// Mitsubishi GX Works2 project: Step Control(end)   PLC: Q01U

PROGRAM conveyor
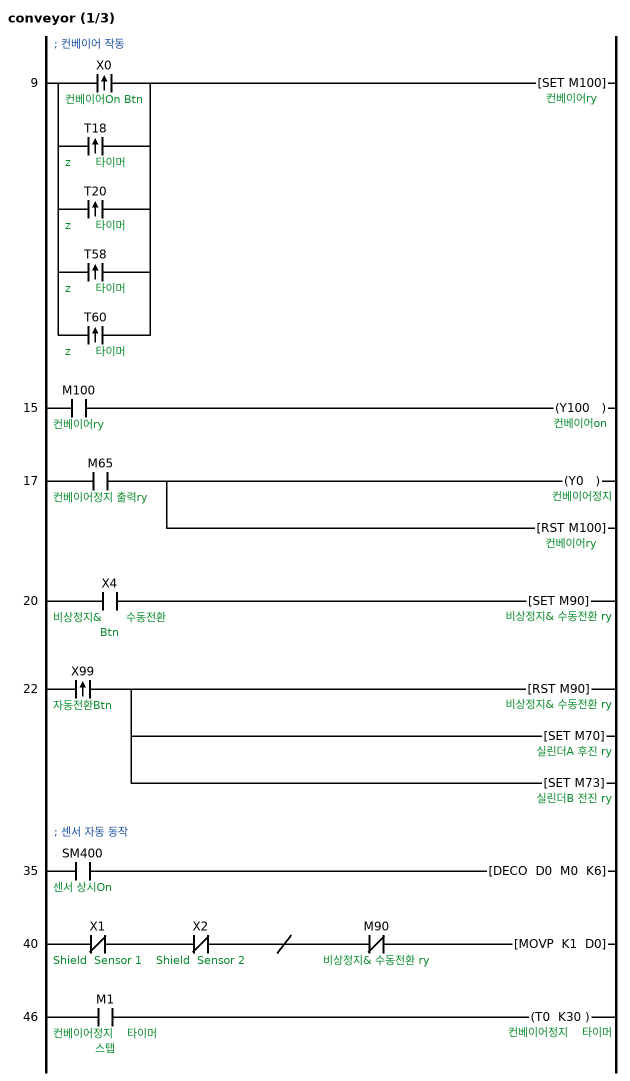
; 컨베이어 작동
9     LDP     X0  ; 컨베이어On Btn
      ORP     T18  ; z       타이머
      ORP     T20  ; z       타이머
      ORP     T58  ; z       타이머
      ORP     T60  ; z       타이머
      SET     M100  ; 컨베이어ry
15    LD      M100  ; 컨베이어ry
      OUT     Y100  ; 컨베이어on
17    LD      M65  ; 컨베이어정지 출력ry
      OUT     Y0  ; 컨베이어정지
      RST     M100  ; 컨베이어ry
20    LD      X4  ; 비상정지&       수동전환 Btn
      SET     M90  ; 비상정지& 수동전환 ry
22    LDP     X99  ; 자동전환Btn
      RST     M90  ; 비상정지& 수동전환 ry
      SET     M70  ; 실린더A 후진 ry
      SET     M73  ; 실린더B 전진 ry
; 센서 자동 동작
35    LD      SM400  ; 센서 상시On
      DECO    D0 M0 K6
40    LDI     X1  ; Shield  Sensor 1
      ANI     X2  ; Shield  Sensor 2
      INV
      ANI     M90  ; 비상정지& 수동전환 ry
      MOVP    K1 D0
46    LD      M1  ; 컨베이어정지    타이머  스탭
      OUT     T0 K30  ; 컨베이어정지    타이머
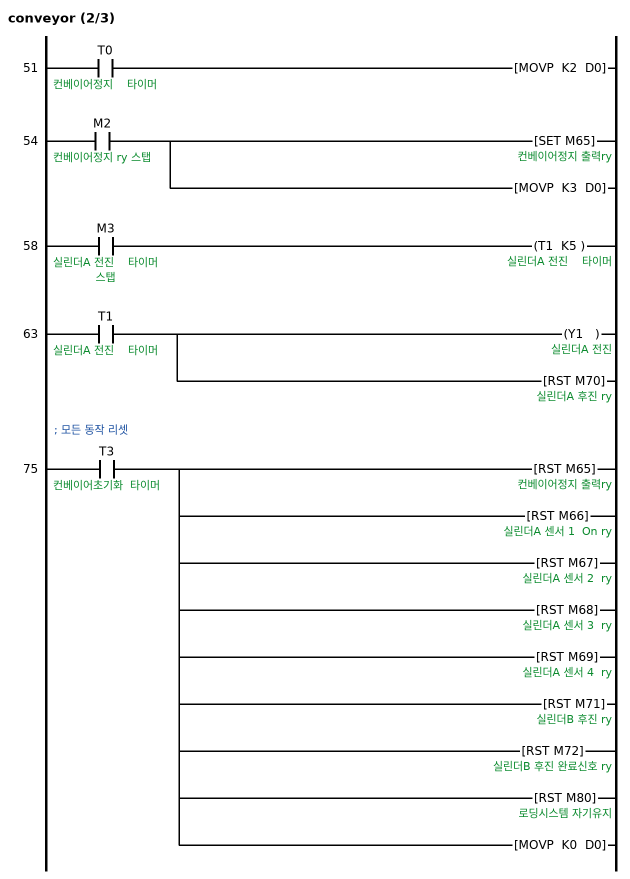
51    LD      T0  ; 컨베이어정지    타이머
      MOVP    K2 D0
54    LD      M2  ; 컨베이어정지 ry 스탭
      SET     M65  ; 컨베이어정지 출력ry
      MOVP    K3 D0
58    LD      M3  ; 실린더A 전진    타이머  스탭
      OUT     T1 K5  ; 실린더A 전진    타이머
63    LD      T1  ; 실린더A 전진    타이머
      OUT     Y1  ; 실린더A 전진
      RST     M70  ; 실린더A 후진 ry
; 모든 동작 리셋
75    LD      T3  ; 컨베이어초기화  타이머
      RST     M65  ; 컨베이어정지 출력ry
      RST     M66  ; 실린더A 센서 1  On ry
      RST     M67  ; 실린더A 센서 2  ry
      RST     M68  ; 실린더A 센서 3  ry
      RST     M69  ; 실린더A 센서 4  ry
      RST     M71  ; 실린더B 후진 ry
      RST     M72  ; 실린더B 후진 완료신호 ry
      RST     M80  ; 로딩시스템 자기유지
      MOVP    K0 D0
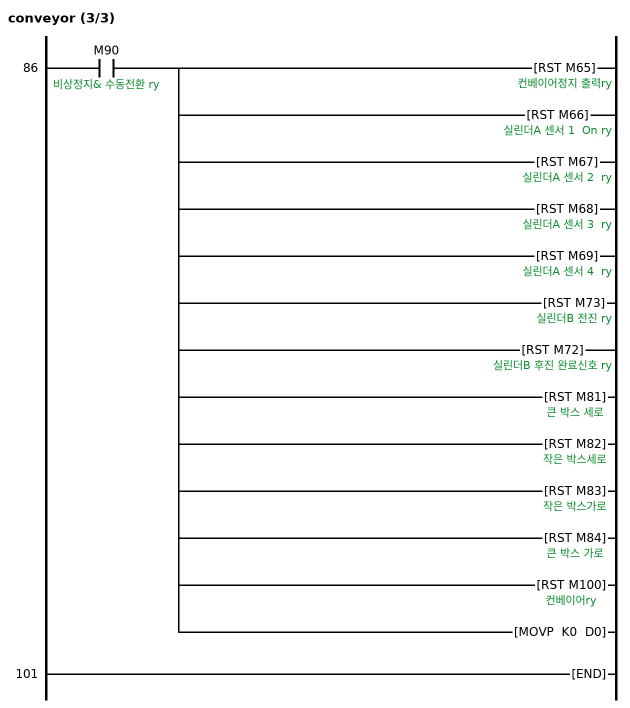
86    LD      M90  ; 비상정지& 수동전환 ry
      RST     M65  ; 컨베이어정지 출력ry
      RST     M66  ; 실린더A 센서 1  On ry
      RST     M67  ; 실린더A 센서 2  ry
      RST     M68  ; 실린더A 센서 3  ry
      RST     M69  ; 실린더A 센서 4  ry
      RST     M73  ; 실린더B 전진 ry
      RST     M72  ; 실린더B 후진 완료신호 ry
      RST     M81  ; 큰 박스 세로
      RST     M82  ; 작은 박스세로
      RST     M83  ; 작은 박스가로
      RST     M84  ; 큰 박스 가로
      RST     M100  ; 컨베이어ry
      MOVP    K0 D0
101   END
END_PROGRAM

PROGRAM cylinder
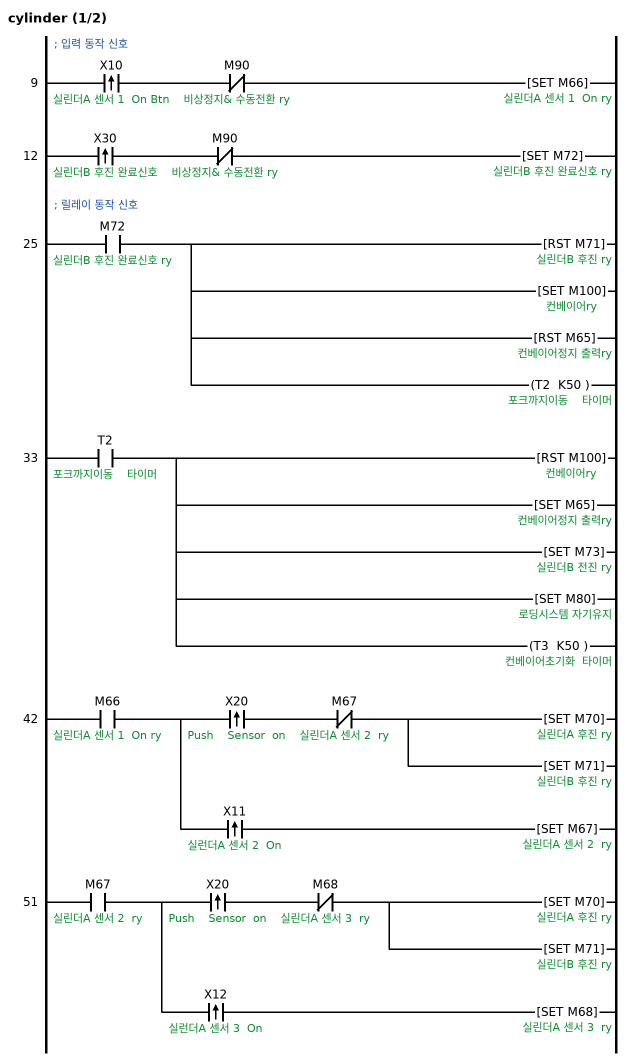
; 입력 동작 신호
9     LDP     X10  ; 실린더A 센서 1  On Btn
      ANI     M90  ; 비상정지& 수동전환 ry
      SET     M66  ; 실린더A 센서 1  On ry
12    LDP     X30  ; 실린더B 후진 완료신호
      ANI     M90  ; 비상정지& 수동전환 ry
      SET     M72  ; 실린더B 후진 완료신호 ry
; 릴레이 동작 신호
25    LD      M72  ; 실린더B 후진 완료신호 ry
      RST     M71  ; 실린더B 후진 ry
      SET     M100  ; 컨베이어ry
      RST     M65  ; 컨베이어정지 출력ry
      OUT     T2 K50  ; 포크까지이동    타이머
33    LD      T2  ; 포크까지이동    타이머
      RST     M100  ; 컨베이어ry
      SET     M65  ; 컨베이어정지 출력ry
      SET     M73  ; 실린더B 전진 ry
      SET     M80  ; 로딩시스템 자기유지
      OUT     T3 K50  ; 컨베이어초기화  타이머
42    LD      M66  ; 실린더A 센서 1  On ry
      MPS
      ANDP    X20  ; Push    Sensor  on
      ANI     M67  ; 실린더A 센서 2  ry
      SET     M70  ; 실린더A 후진 ry
      SET     M71  ; 실린더B 후진 ry
      MPP
      ANDP    X11  ; 실런더A 센서 2  On
      SET     M67  ; 실린더A 센서 2  ry
51    LD      M67  ; 실린더A 센서 2  ry
      MPS
      ANDP    X20  ; Push    Sensor  on
      ANI     M68  ; 실린더A 센서 3  ry
      SET     M70  ; 실린더A 후진 ry
      SET     M71  ; 실린더B 후진 ry
      MPP
      ANDP    X12  ; 실런더A 센서 3  On
      SET     M68  ; 실린더A 센서 3  ry
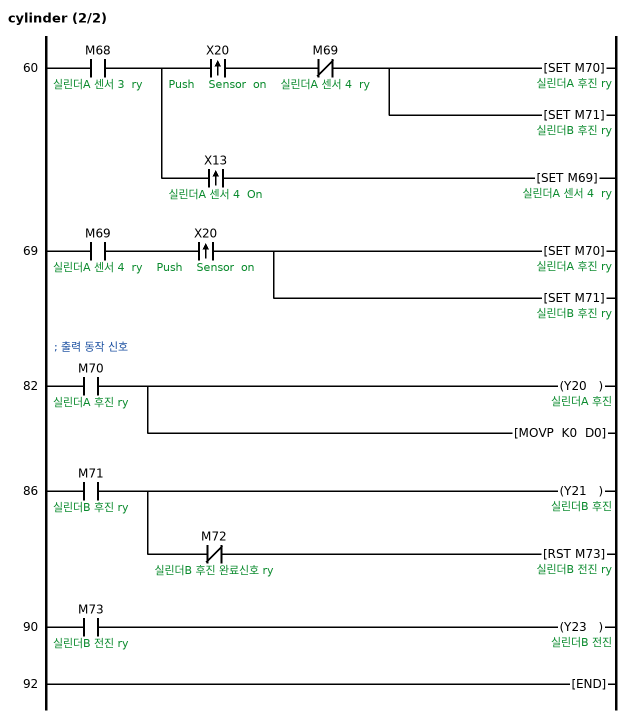
60    LD      M68  ; 실린더A 센서 3  ry
      MPS
      ANDP    X20  ; Push    Sensor  on
      ANI     M69  ; 실린더A 센서 4  ry
      SET     M70  ; 실린더A 후진 ry
      SET     M71  ; 실린더B 후진 ry
      MPP
      ANDP    X13  ; 실린더A 센서 4  On
      SET     M69  ; 실린더A 센서 4  ry
69    LD      M69  ; 실린더A 센서 4  ry
      ANDP    X20  ; Push    Sensor  on
      SET     M70  ; 실린더A 후진 ry
      SET     M71  ; 실린더B 후진 ry
; 출력 동작 신호
82    LD      M70  ; 실린더A 후진 ry
      OUT     Y20  ; 실린더A 후진
      MOVP    K0 D0
86    LD      M71  ; 실린더B 후진 ry
      OUT     Y21  ; 실린더B 후진
      ANI     M72  ; 실린더B 후진 완료신호 ry
      RST     M73  ; 실린더B 전진 ry
90    LD      M73  ; 실린더B 전진 ry
      OUT     Y23  ; 실린더B 전진
92    END
END_PROGRAM

PROGRAM manual
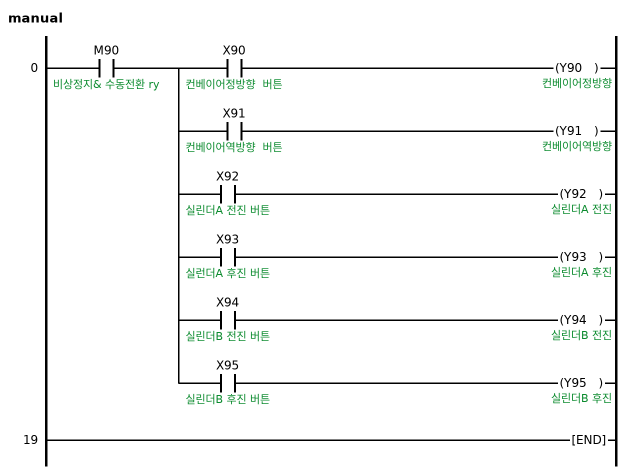
0     LD      M90  ; 비상정지& 수동전환 ry
      MPS
      AND     X90  ; 컨베이어정방향  버튼
      OUT     Y90  ; 컨베이어정방향
      MRD
      AND     X91  ; 컨베이어역방향  버튼
      OUT     Y91  ; 컨베이어역방향
      MRD
      AND     X92  ; 실린더A 전진 버튼
      OUT     Y92  ; 실린더A 전진
      MRD
      AND     X93  ; 실런더A 후진 버튼
      OUT     Y93  ; 실린더A 후진
      MRD
      AND     X94  ; 실린더B 전진 버튼
      OUT     Y94  ; 실린더B 전진
      MPP
      AND     X95  ; 실린더B 후진 버튼
      OUT     Y95  ; 실린더B 후진
19    END
END_PROGRAM

PROGRAM boxSize
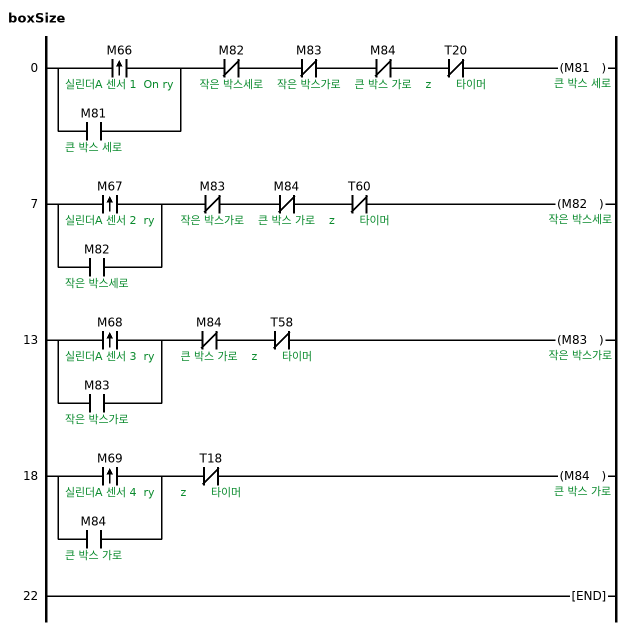
0     LDP     M66  ; 실린더A 센서 1  On ry
      OR      M81  ; 큰 박스 세로
      ANI     M82  ; 작은 박스세로
      ANI     M83  ; 작은 박스가로
      ANI     M84  ; 큰 박스 가로
      ANI     T20  ; z       타이머
      OUT     M81  ; 큰 박스 세로
7     LDP     M67  ; 실린더A 센서 2  ry
      OR      M82  ; 작은 박스세로
      ANI     M83  ; 작은 박스가로
      ANI     M84  ; 큰 박스 가로
      ANI     T60  ; z       타이머
      OUT     M82  ; 작은 박스세로
13    LDP     M68  ; 실린더A 센서 3  ry
      OR      M83  ; 작은 박스가로
      ANI     M84  ; 큰 박스 가로
      ANI     T58  ; z       타이머
      OUT     M83  ; 작은 박스가로
18    LDP     M69  ; 실린더A 센서 4  ry
      OR      M84  ; 큰 박스 가로
      ANI     T18  ; z       타이머
      OUT     M84  ; 큰 박스 가로
22    END
END_PROGRAM

PROGRAM Box4move
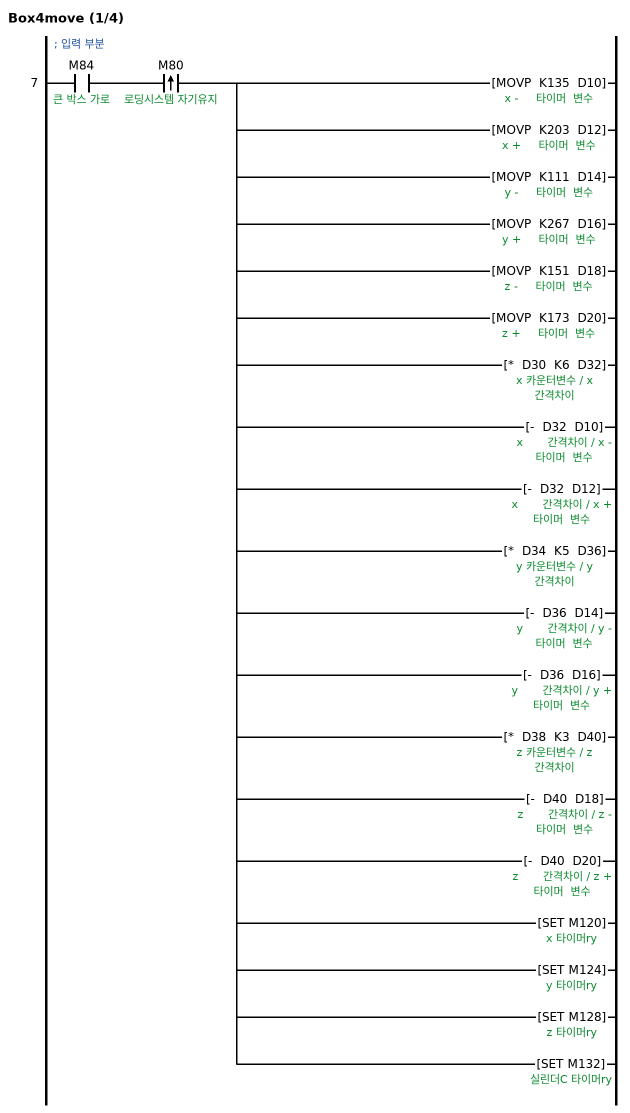
; 입력 부분
7     LD      M84  ; 큰 박스 가로
      ANDP    M80  ; 로딩시스템 자기유지
      MOVP    K135 D10  ; x -     타이머  변수
      MOVP    K203 D12  ; x +     타이머  변수
      MOVP    K111 D14  ; y -     타이머  변수
      MOVP    K267 D16  ; y +     타이머  변수
      MOVP    K151 D18  ; z -     타이머  변수
      MOVP    K173 D20  ; z +     타이머  변수
      *       D30 K6 D32  ; x 카운터변수 / x       간격차이
      -       D32 D10
      -       D32 D12
      *       D34 K5 D36  ; y 카운터변수 / y       간격차이
      -       D36 D14
      -       D36 D16
      *       D38 K3 D40  ; z 카운터변수 / z       간격차이
      -       D40 D18
      -       D40 D20
      SET     M120  ; x 타이머ry
      SET     M124  ; y 타이머ry
      SET     M128  ; z 타이머ry
      SET     M132  ; 실린더C 타이머ry
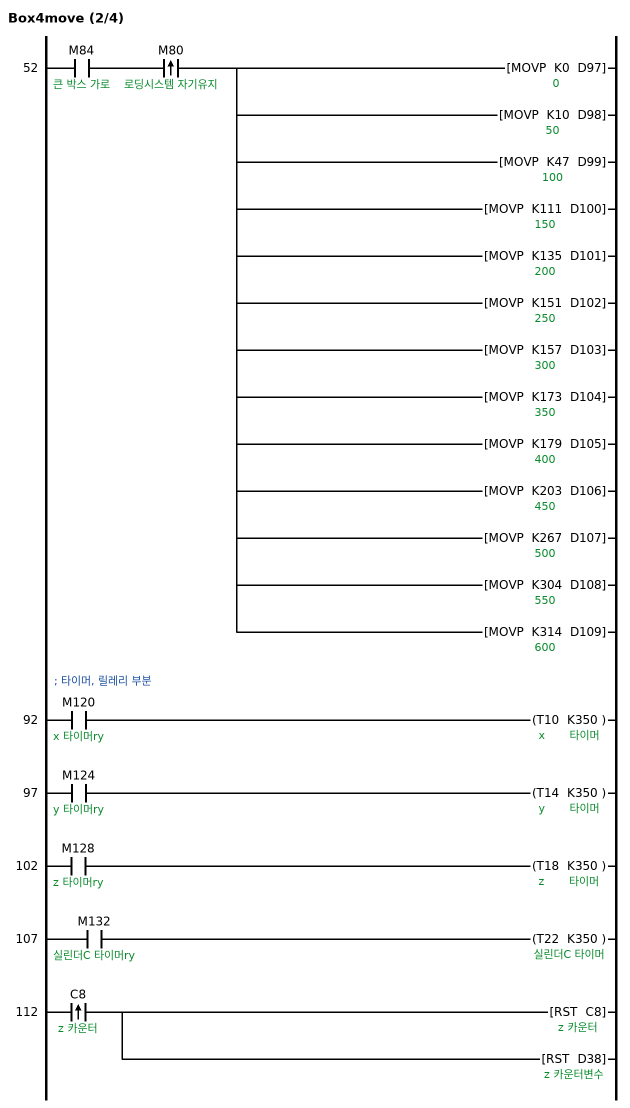
52    LD      M84  ; 큰 박스 가로
      ANDP    M80  ; 로딩시스템 자기유지
      MOVP    K0 D97  ; 0
      MOVP    K10 D98  ; 50
      MOVP    K47 D99  ; 100
      MOVP    K111 D100  ; 150
      MOVP    K135 D101  ; 200
      MOVP    K151 D102  ; 250
      MOVP    K157 D103  ; 300
      MOVP    K173 D104  ; 350
      MOVP    K179 D105  ; 400
      MOVP    K203 D106  ; 450
      MOVP    K267 D107  ; 500
      MOVP    K304 D108  ; 550
      MOVP    K314 D109  ; 600
; 타이머, 릴레리 부분
92    LD      M120  ; x 타이머ry
      OUT     T10 K350  ; x       타이머
97    LD      M124  ; y 타이머ry
      OUT     T14 K350  ; y       타이머
102   LD      M128  ; z 타이머ry
      OUT     T18 K350  ; z       타이머
107   LD      M132  ; 실린더C 타이머ry
      OUT     T22 K350  ; 실린더C 타이머
112   LDP     C8  ; z 카운터
      RST     C8  ; z 카운터
      RST     D38  ; z 카운터변수
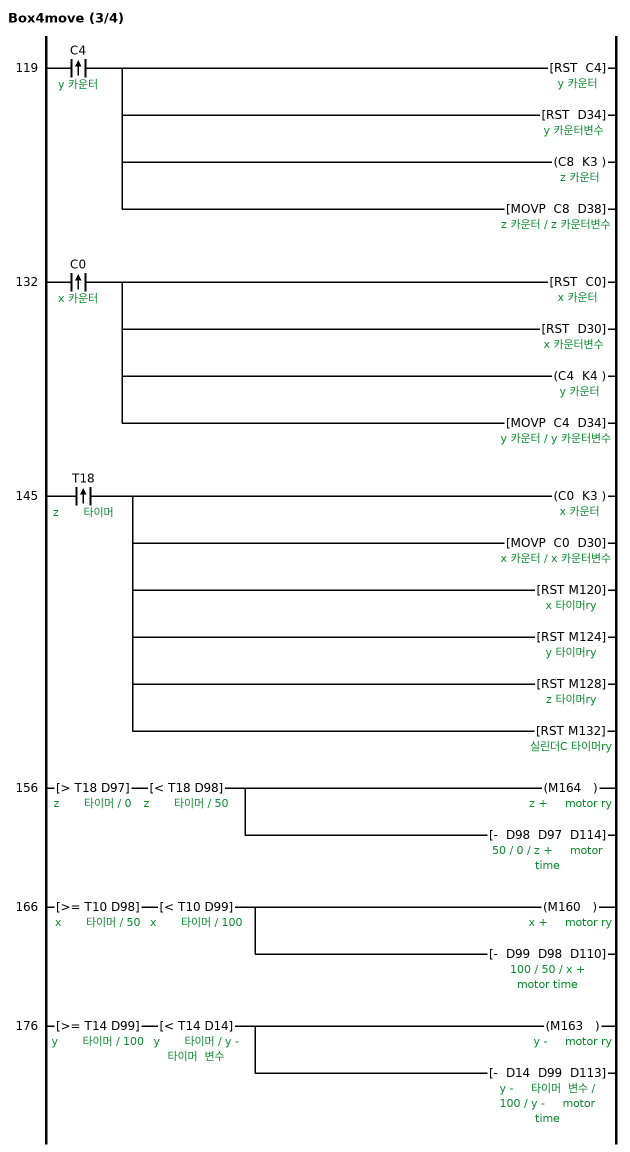
119   LDP     C4  ; y 카운터
      RST     C4  ; y 카운터
      RST     D34  ; y 카운터변수
      OUT     C8 K3  ; z 카운터
      MOVP    C8 D38
132   LDP     C0  ; x 카운터
      RST     C0  ; x 카운터
      RST     D30  ; x 카운터변수
      OUT     C4 K4  ; y 카운터
      MOVP    C4 D34
145   LDP     T18  ; z       타이머
      OUT     C0 K3  ; x 카운터
      MOVP    C0 D30
      RST     M120  ; x 타이머ry
      RST     M124  ; y 타이머ry
      RST     M128  ; z 타이머ry
      RST     M132  ; 실린더C 타이머ry
156   LD>     T18 D97  ; z       타이머 / 0
      AND<    T18 D98  ; z       타이머 / 50
      OUT     M164  ; z +     motor ry
      -       D98 D97 D114  ; z +     motor time
166   LD>=    T10 D98  ; x       타이머 / 50
      AND<    T10 D99  ; x       타이머 / 100
      OUT     M160  ; x +     motor ry
      -       D99 D98 D110  ; x +     motor time
176   LD>=    T14 D99  ; y       타이머 / 100
      AND<    T14 D14  ; y       타이머 / y -     타이머  변수
      OUT     M163  ; y -     motor ry
      -       D14 D99 D113  ; y -     motor time
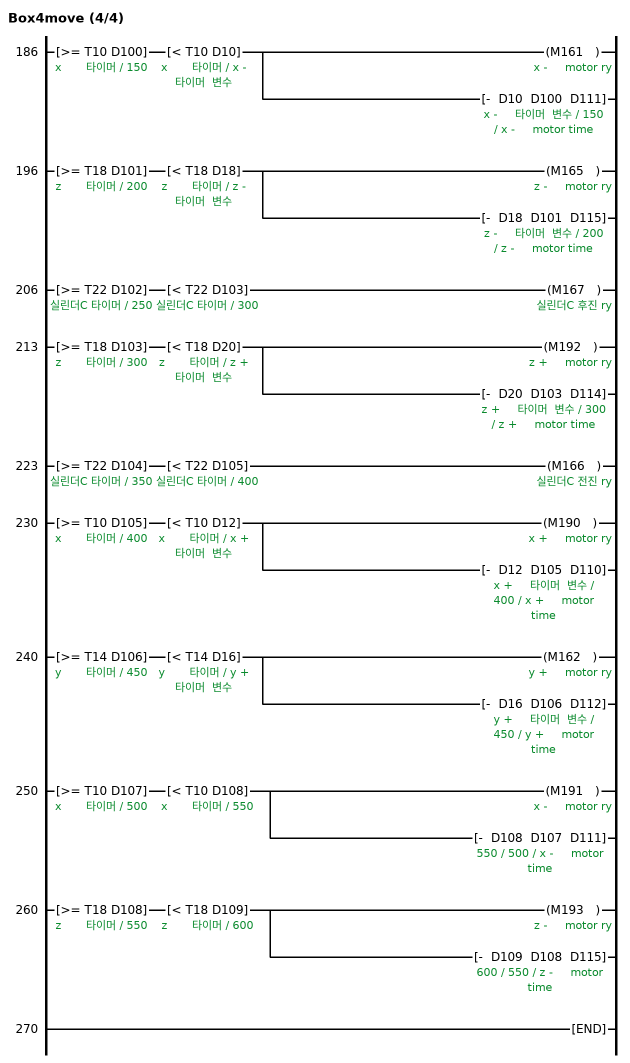
186   LD>=    T10 D100  ; x       타이머 / 150
      AND<    T10 D10  ; x       타이머 / x -     타이머  변수
      OUT     M161  ; x -     motor ry
      -       D10 D100 D111  ; x -     motor time
196   LD>=    T18 D101  ; z       타이머 / 200
      AND<    T18 D18  ; z       타이머 / z -     타이머  변수
      OUT     M165  ; z -     motor ry
      -       D18 D101 D115  ; z -     motor time
206   LD>=    T22 D102  ; 실린더C 타이머 / 250
      AND<    T22 D103  ; 실린더C 타이머 / 300
      OUT     M167  ; 실린더C 후진 ry
213   LD>=    T18 D103  ; z       타이머 / 300
      AND<    T18 D20  ; z       타이머 / z +     타이머  변수
      OUT     M192  ; z +     motor ry
      -       D20 D103 D114
223   LD>=    T22 D104  ; 실린더C 타이머 / 350
      AND<    T22 D105  ; 실린더C 타이머 / 400
      OUT     M166  ; 실린더C 전진 ry
230   LD>=    T10 D105  ; x       타이머 / 400
      AND<    T10 D12  ; x       타이머 / x +     타이머  변수
      OUT     M190  ; x +     motor ry
      -       D12 D105 D110
240   LD>=    T14 D106  ; y       타이머 / 450
      AND<    T14 D16  ; y       타이머 / y +     타이머  변수
      OUT     M162  ; y +     motor ry
      -       D16 D106 D112  ; y +     motor time
250   LD>=    T10 D107  ; x       타이머 / 500
      AND<    T10 D108  ; x       타이머 / 550
      OUT     M191  ; x -     motor ry
      -       D108 D107 D111
260   LD>=    T18 D108  ; z       타이머 / 550
      AND<    T18 D109  ; z       타이머 / 600
      OUT     M193  ; z -     motor ry
      -       D109 D108 D115
270   END
END_PROGRAM

PROGRAM Lmanual
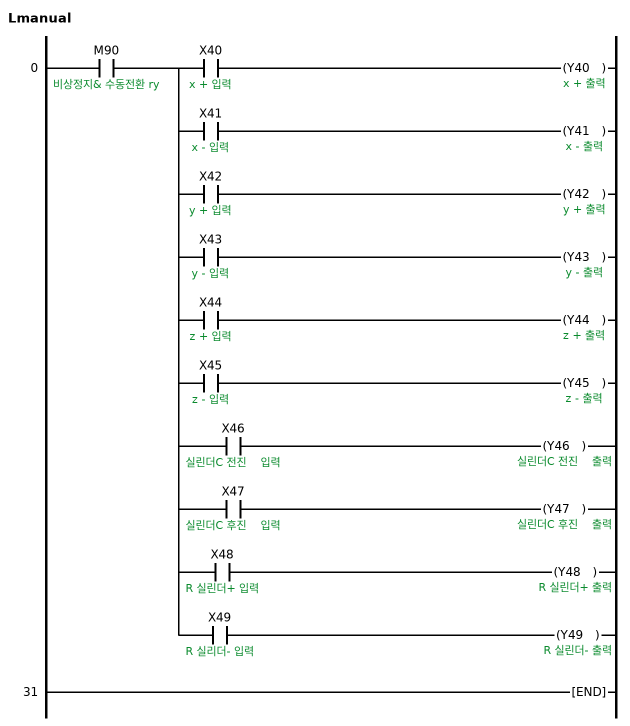
0     LD      M90  ; 비상정지& 수동전환 ry
      MPS
      AND     X40  ; x + 입력
      OUT     Y40  ; x + 출력
      MRD
      AND     X41  ; x - 입력
      OUT     Y41  ; x - 출력
      MRD
      AND     X42  ; y + 입력
      OUT     Y42  ; y + 출력
      MRD
      AND     X43  ; y - 입력
      OUT     Y43  ; y - 출력
      MRD
      AND     X44  ; z + 입력
      OUT     Y44  ; z + 출력
      MRD
      AND     X45  ; z - 입력
      OUT     Y45  ; z - 출력
      MRD
      AND     X46  ; 실린더C 전진    입력
      OUT     Y46  ; 실린더C 전진    출력
      MRD
      AND     X47  ; 실린더C 후진    입력
      OUT     Y47  ; 실린더C 후진    출력
      MRD
      AND     X48  ; R 실린더+ 입력
      OUT     Y48  ; R 실린더+ 출력
      MPP
      AND     X49  ; R 실리더- 입력
      OUT     Y49  ; R 실린더- 출력
31    END
END_PROGRAM

PROGRAM Box1move
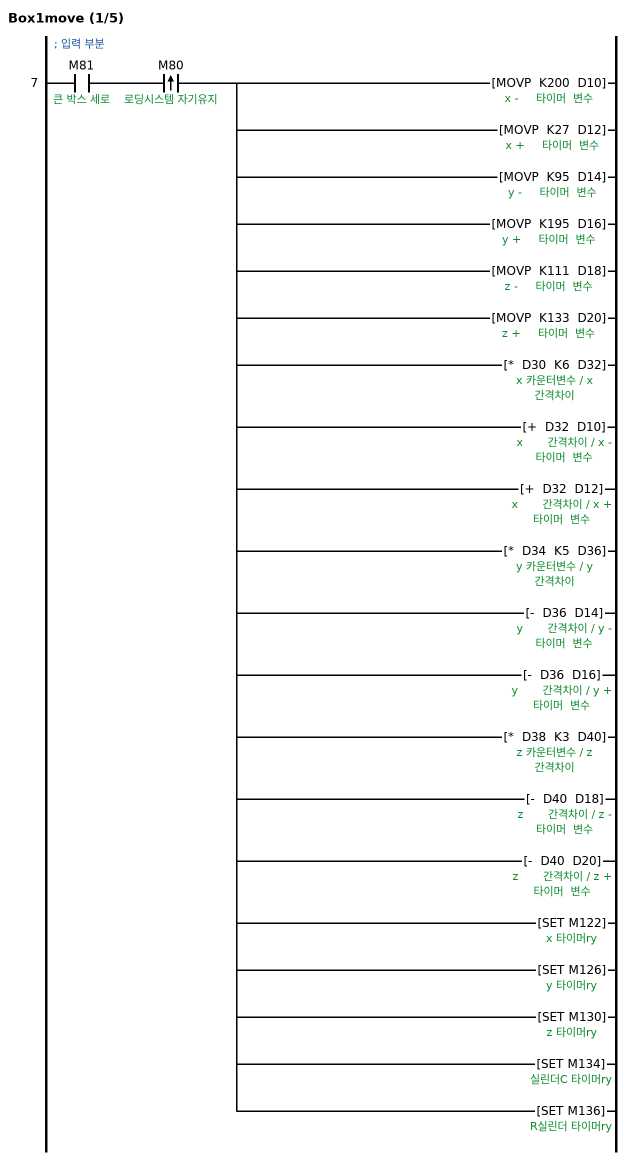
; 입력 부분
7     LD      M81  ; 큰 박스 세로
      ANDP    M80  ; 로딩시스템 자기유지
      MOVP    K200 D10  ; x -     타이머  변수
      MOVP    K27 D12  ; x +     타이머  변수
      MOVP    K95 D14  ; y -     타이머  변수
      MOVP    K195 D16  ; y +     타이머  변수
      MOVP    K111 D18  ; z -     타이머  변수
      MOVP    K133 D20  ; z +     타이머  변수
      *       D30 K6 D32  ; x 카운터변수 / x       간격차이
      +       D32 D10
      +       D32 D12
      *       D34 K5 D36  ; y 카운터변수 / y       간격차이
      -       D36 D14
      -       D36 D16
      *       D38 K3 D40  ; z 카운터변수 / z       간격차이
      -       D40 D18
      -       D40 D20
      SET     M122  ; x 타이머ry
      SET     M126  ; y 타이머ry
      SET     M130  ; z 타이머ry
      SET     M134  ; 실린더C 타이머ry
      SET     M136  ; R실린더 타이머ry
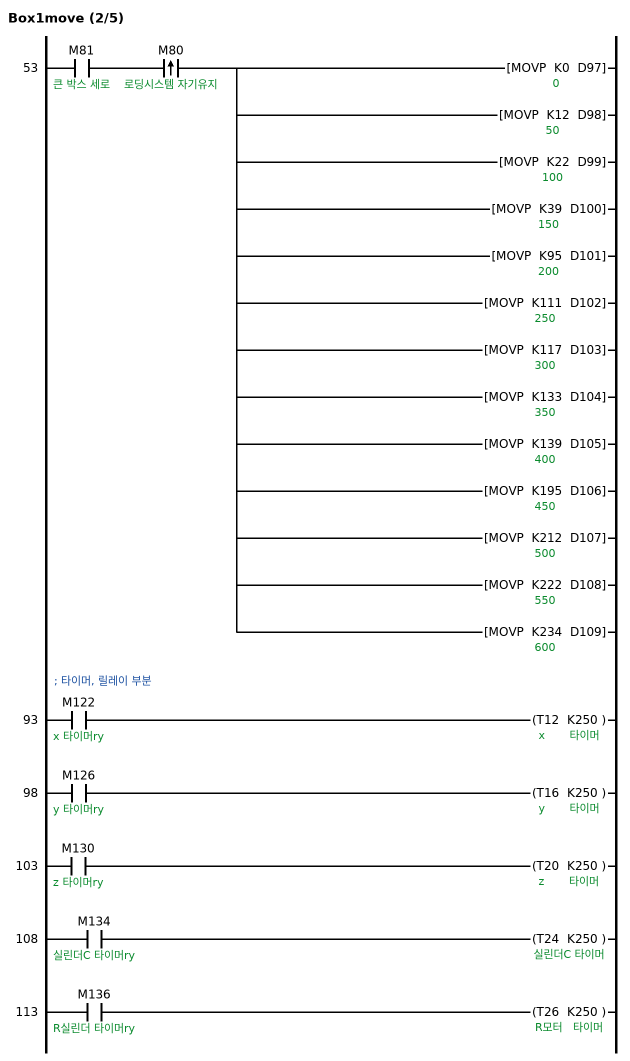
53    LD      M81  ; 큰 박스 세로
      ANDP    M80  ; 로딩시스템 자기유지
      MOVP    K0 D97  ; 0
      MOVP    K12 D98  ; 50
      MOVP    K22 D99  ; 100
      MOVP    K39 D100  ; 150
      MOVP    K95 D101  ; 200
      MOVP    K111 D102  ; 250
      MOVP    K117 D103  ; 300
      MOVP    K133 D104  ; 350
      MOVP    K139 D105  ; 400
      MOVP    K195 D106  ; 450
      MOVP    K212 D107  ; 500
      MOVP    K222 D108  ; 550
      MOVP    K234 D109  ; 600
; 타이머, 릴레이 부분
93    LD      M122  ; x 타이머ry
      OUT     T12 K250  ; x       타이머
98    LD      M126  ; y 타이머ry
      OUT     T16 K250  ; y       타이머
103   LD      M130  ; z 타이머ry
      OUT     T20 K250  ; z       타이머
108   LD      M134  ; 실린더C 타이머ry
      OUT     T24 K250  ; 실린더C 타이머
113   LD      M136  ; R실린더 타이머ry
      OUT     T26 K250  ; R모터   타이머
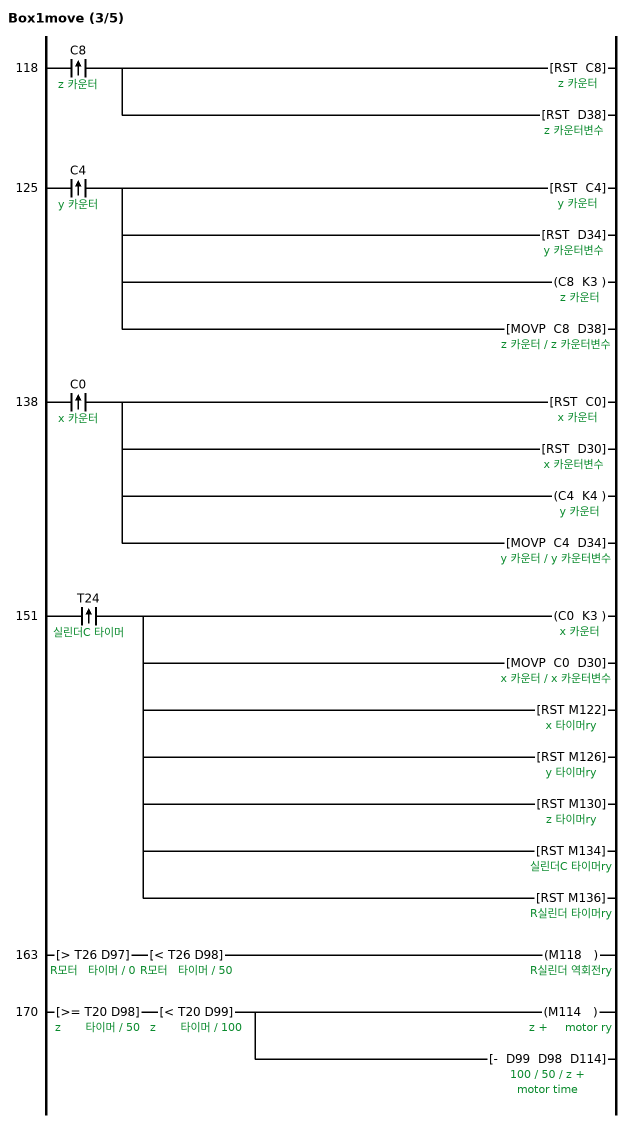
118   LDP     C8  ; z 카운터
      RST     C8  ; z 카운터
      RST     D38  ; z 카운터변수
125   LDP     C4  ; y 카운터
      RST     C4  ; y 카운터
      RST     D34  ; y 카운터변수
      OUT     C8 K3  ; z 카운터
      MOVP    C8 D38
138   LDP     C0  ; x 카운터
      RST     C0  ; x 카운터
      RST     D30  ; x 카운터변수
      OUT     C4 K4  ; y 카운터
      MOVP    C4 D34
151   LDP     T24  ; 실린더C 타이머
      OUT     C0 K3  ; x 카운터
      MOVP    C0 D30
      RST     M122  ; x 타이머ry
      RST     M126  ; y 타이머ry
      RST     M130  ; z 타이머ry
      RST     M134  ; 실린더C 타이머ry
      RST     M136  ; R실린더 타이머ry
163   LD>     T26 D97  ; R모터   타이머 / 0
      AND<    T26 D98  ; R모터   타이머 / 50
      OUT     M118  ; R실린더 역회전ry
170   LD>=    T20 D98  ; z       타이머 / 50
      AND<    T20 D99  ; z       타이머 / 100
      OUT     M114  ; z +     motor ry
      -       D99 D98 D114  ; z +     motor time
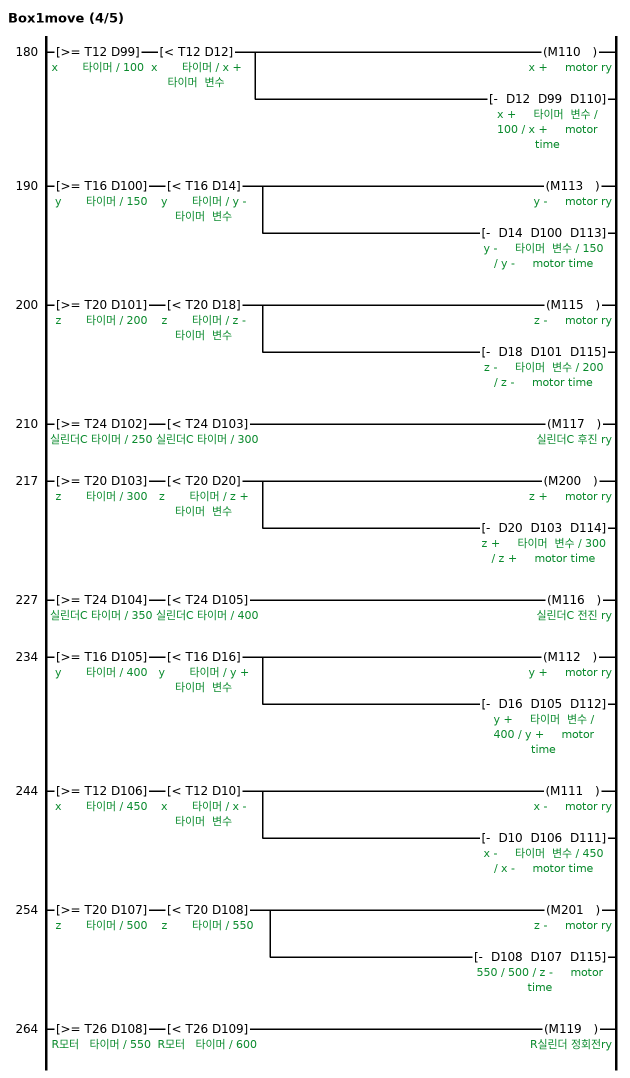
180   LD>=    T12 D99  ; x       타이머 / 100
      AND<    T12 D12  ; x       타이머 / x +     타이머  변수
      OUT     M110  ; x +     motor ry
      -       D12 D99 D110  ; x +     motor time
190   LD>=    T16 D100  ; y       타이머 / 150
      AND<    T16 D14  ; y       타이머 / y -     타이머  변수
      OUT     M113  ; y -     motor ry
      -       D14 D100 D113  ; y -     motor time
200   LD>=    T20 D101  ; z       타이머 / 200
      AND<    T20 D18  ; z       타이머 / z -     타이머  변수
      OUT     M115  ; z -     motor ry
      -       D18 D101 D115  ; z -     motor time
210   LD>=    T24 D102  ; 실린더C 타이머 / 250
      AND<    T24 D103  ; 실린더C 타이머 / 300
      OUT     M117  ; 실린더C 후진 ry
217   LD>=    T20 D103  ; z       타이머 / 300
      AND<    T20 D20  ; z       타이머 / z +     타이머  변수
      OUT     M200  ; z +     motor ry
      -       D20 D103 D114
227   LD>=    T24 D104  ; 실린더C 타이머 / 350
      AND<    T24 D105  ; 실린더C 타이머 / 400
      OUT     M116  ; 실린더C 전진 ry
234   LD>=    T16 D105  ; y       타이머 / 400
      AND<    T16 D16  ; y       타이머 / y +     타이머  변수
      OUT     M112  ; y +     motor ry
      -       D16 D105 D112  ; y +     motor time
244   LD>=    T12 D106  ; x       타이머 / 450
      AND<    T12 D10  ; x       타이머 / x -     타이머  변수
      OUT     M111  ; x -     motor ry
      -       D10 D106 D111  ; x -     motor time
254   LD>=    T20 D107  ; z       타이머 / 500
      AND<    T20 D108  ; z       타이머 / 550
      OUT     M201  ; z -     motor ry
      -       D108 D107 D115
264   LD>=    T26 D108  ; R모터   타이머 / 550
      AND<    T26 D109  ; R모터   타이머 / 600
      OUT     M119  ; R실린더 정회전ry
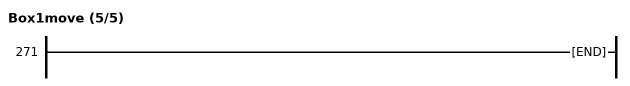
271   END
END_PROGRAM

PROGRAM Box2move
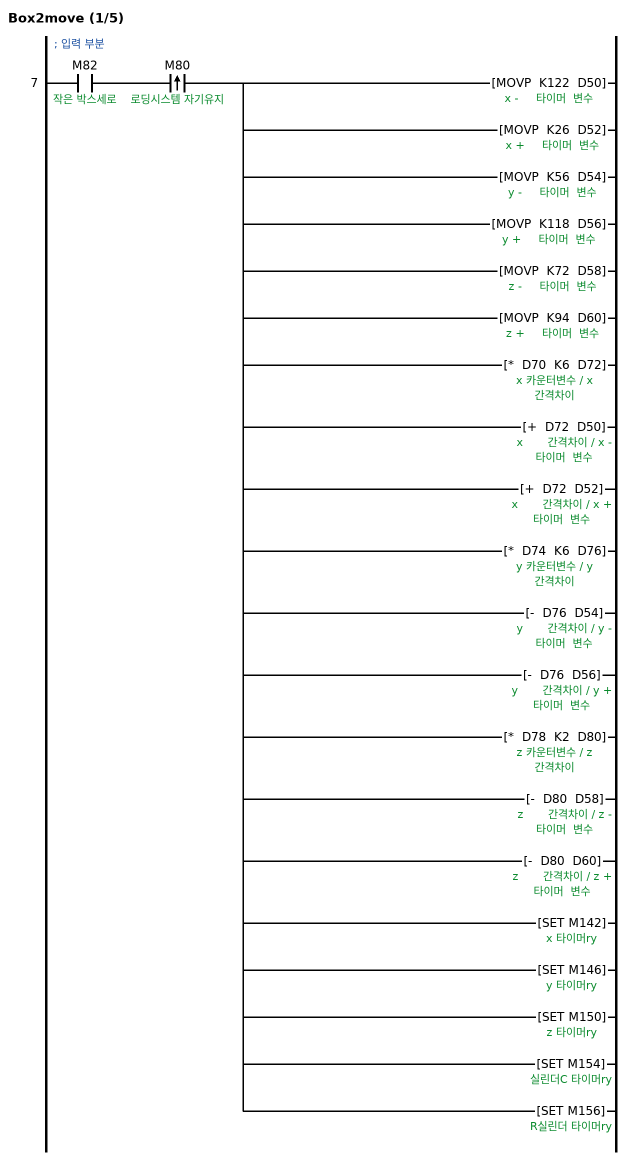
; 입력 부분
7     LD      M82  ; 작은 박스세로
      ANDP    M80  ; 로딩시스템 자기유지
      MOVP    K122 D50  ; x -     타이머  변수
      MOVP    K26 D52  ; x +     타이머  변수
      MOVP    K56 D54  ; y -     타이머  변수
      MOVP    K118 D56  ; y +     타이머  변수
      MOVP    K72 D58  ; z -     타이머  변수
      MOVP    K94 D60  ; z +     타이머  변수
      *       D70 K6 D72  ; x 카운터변수 / x       간격차이
      +       D72 D50
      +       D72 D52
      *       D74 K6 D76  ; y 카운터변수 / y       간격차이
      -       D76 D54
      -       D76 D56
      *       D78 K2 D80  ; z 카운터변수 / z       간격차이
      -       D80 D58
      -       D80 D60
      SET     M142  ; x 타이머ry
      SET     M146  ; y 타이머ry
      SET     M150  ; z 타이머ry
      SET     M154  ; 실린더C 타이머ry
      SET     M156  ; R실린더 타이머ry
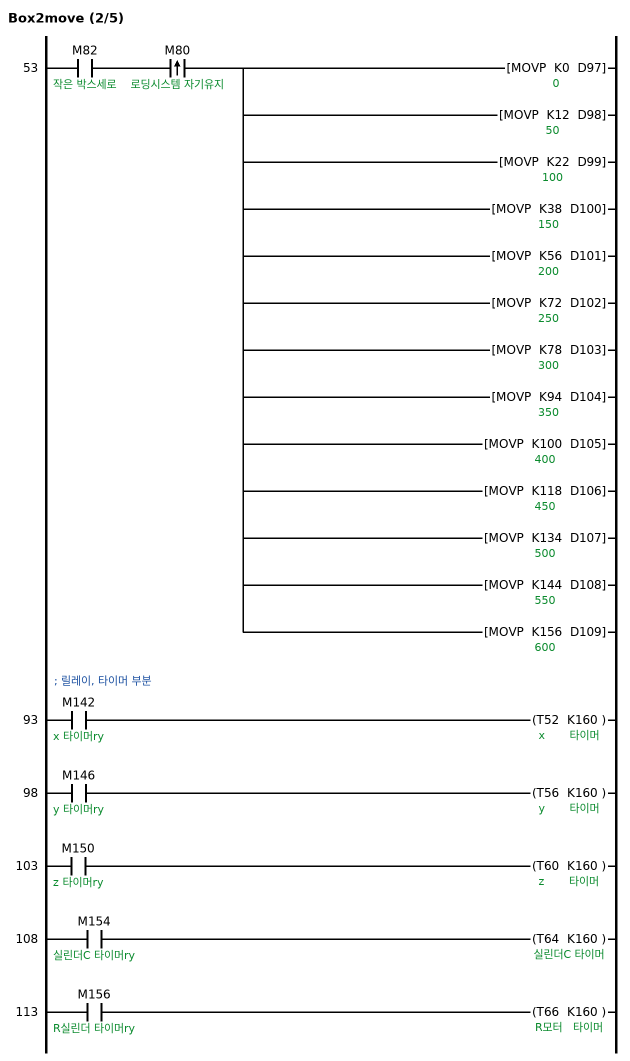
53    LD      M82  ; 작은 박스세로
      ANDP    M80  ; 로딩시스템 자기유지
      MOVP    K0 D97  ; 0
      MOVP    K12 D98  ; 50
      MOVP    K22 D99  ; 100
      MOVP    K38 D100  ; 150
      MOVP    K56 D101  ; 200
      MOVP    K72 D102  ; 250
      MOVP    K78 D103  ; 300
      MOVP    K94 D104  ; 350
      MOVP    K100 D105  ; 400
      MOVP    K118 D106  ; 450
      MOVP    K134 D107  ; 500
      MOVP    K144 D108  ; 550
      MOVP    K156 D109  ; 600
; 릴레이, 타이머 부분
93    LD      M142  ; x 타이머ry
      OUT     T52 K160  ; x       타이머
98    LD      M146  ; y 타이머ry
      OUT     T56 K160  ; y       타이머
103   LD      M150  ; z 타이머ry
      OUT     T60 K160  ; z       타이머
108   LD      M154  ; 실린더C 타이머ry
      OUT     T64 K160  ; 실린더C 타이머
113   LD      M156  ; R실린더 타이머ry
      OUT     T66 K160  ; R모터   타이머
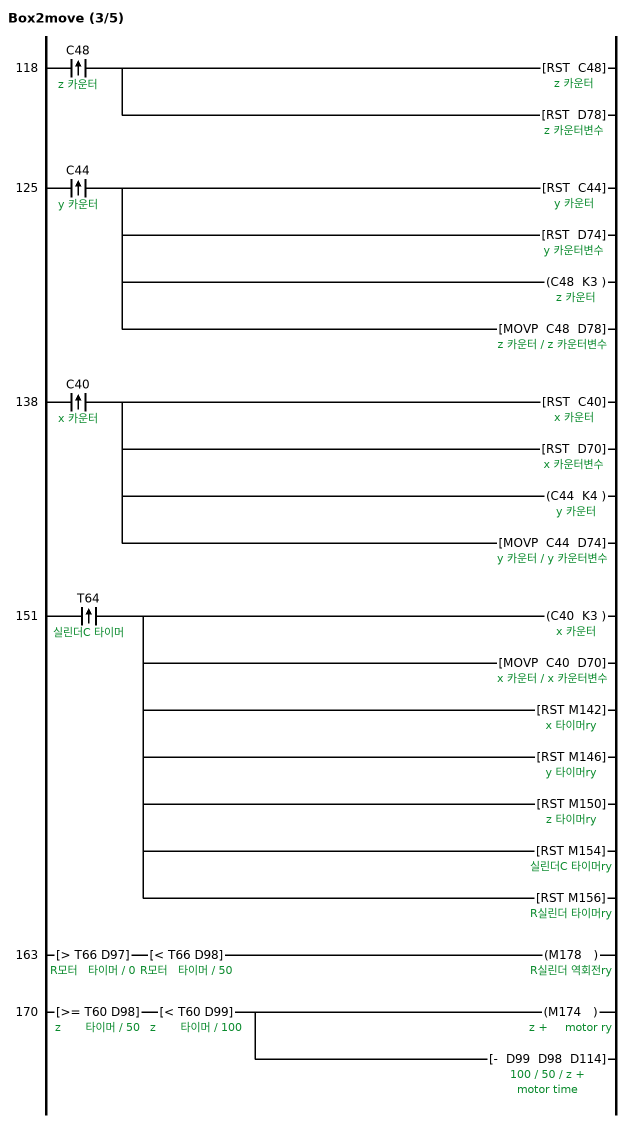
118   LDP     C48  ; z 카운터
      RST     C48  ; z 카운터
      RST     D78  ; z 카운터변수
125   LDP     C44  ; y 카운터
      RST     C44  ; y 카운터
      RST     D74  ; y 카운터변수
      OUT     C48 K3  ; z 카운터
      MOVP    C48 D78
138   LDP     C40  ; x 카운터
      RST     C40  ; x 카운터
      RST     D70  ; x 카운터변수
      OUT     C44 K4  ; y 카운터
      MOVP    C44 D74
151   LDP     T64  ; 실린더C 타이머
      OUT     C40 K3  ; x 카운터
      MOVP    C40 D70
      RST     M142  ; x 타이머ry
      RST     M146  ; y 타이머ry
      RST     M150  ; z 타이머ry
      RST     M154  ; 실린더C 타이머ry
      RST     M156  ; R실린더 타이머ry
163   LD>     T66 D97  ; R모터   타이머 / 0
      AND<    T66 D98  ; R모터   타이머 / 50
      OUT     M178  ; R실린더 역회전ry
170   LD>=    T60 D98  ; z       타이머 / 50
      AND<    T60 D99  ; z       타이머 / 100
      OUT     M174  ; z +     motor ry
      -       D99 D98 D114  ; z +     motor time
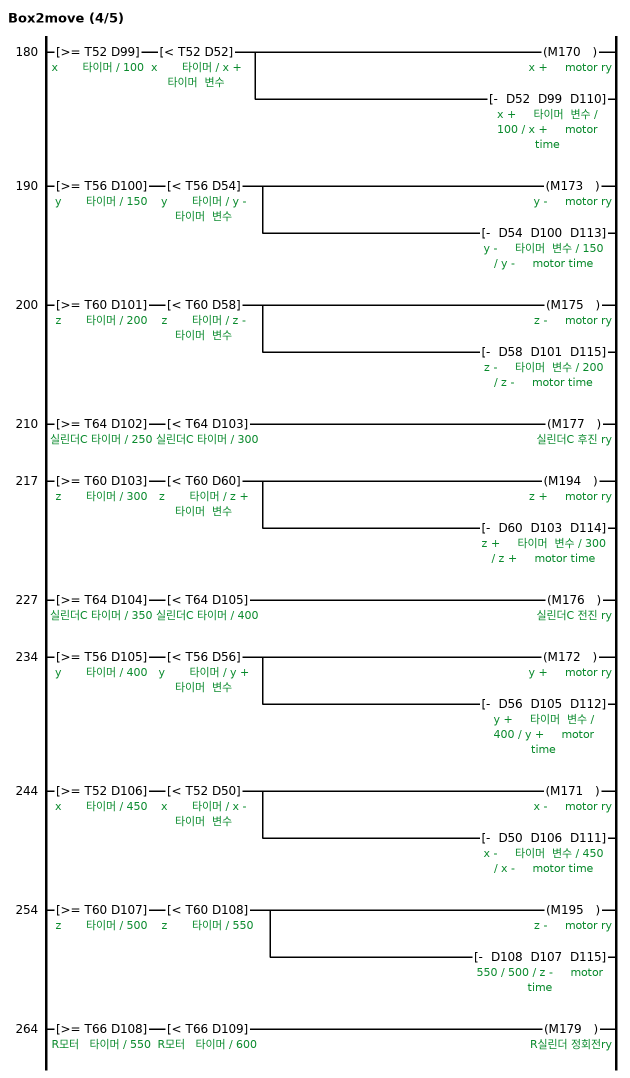
180   LD>=    T52 D99  ; x       타이머 / 100
      AND<    T52 D52  ; x       타이머 / x +     타이머  변수
      OUT     M170  ; x +     motor ry
      -       D52 D99 D110  ; x +     motor time
190   LD>=    T56 D100  ; y       타이머 / 150
      AND<    T56 D54  ; y       타이머 / y -     타이머  변수
      OUT     M173  ; y -     motor ry
      -       D54 D100 D113  ; y -     motor time
200   LD>=    T60 D101  ; z       타이머 / 200
      AND<    T60 D58  ; z       타이머 / z -     타이머  변수
      OUT     M175  ; z -     motor ry
      -       D58 D101 D115  ; z -     motor time
210   LD>=    T64 D102  ; 실린더C 타이머 / 250
      AND<    T64 D103  ; 실린더C 타이머 / 300
      OUT     M177  ; 실린더C 후진 ry
217   LD>=    T60 D103  ; z       타이머 / 300
      AND<    T60 D60  ; z       타이머 / z +     타이머  변수
      OUT     M194  ; z +     motor ry
      -       D60 D103 D114
227   LD>=    T64 D104  ; 실린더C 타이머 / 350
      AND<    T64 D105  ; 실린더C 타이머 / 400
      OUT     M176  ; 실린더C 전진 ry
234   LD>=    T56 D105  ; y       타이머 / 400
      AND<    T56 D56  ; y       타이머 / y +     타이머  변수
      OUT     M172  ; y +     motor ry
      -       D56 D105 D112  ; y +     motor time
244   LD>=    T52 D106  ; x       타이머 / 450
      AND<    T52 D50  ; x       타이머 / x -     타이머  변수
      OUT     M171  ; x -     motor ry
      -       D50 D106 D111  ; x -     motor time
254   LD>=    T60 D107  ; z       타이머 / 500
      AND<    T60 D108  ; z       타이머 / 550
      OUT     M195  ; z -     motor ry
      -       D108 D107 D115
264   LD>=    T66 D108  ; R모터   타이머 / 550
      AND<    T66 D109  ; R모터   타이머 / 600
      OUT     M179  ; R실린더 정회전ry
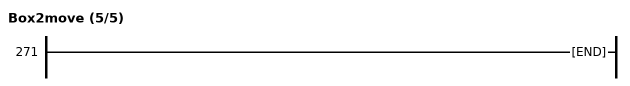
271   END
END_PROGRAM

PROGRAM Box3move
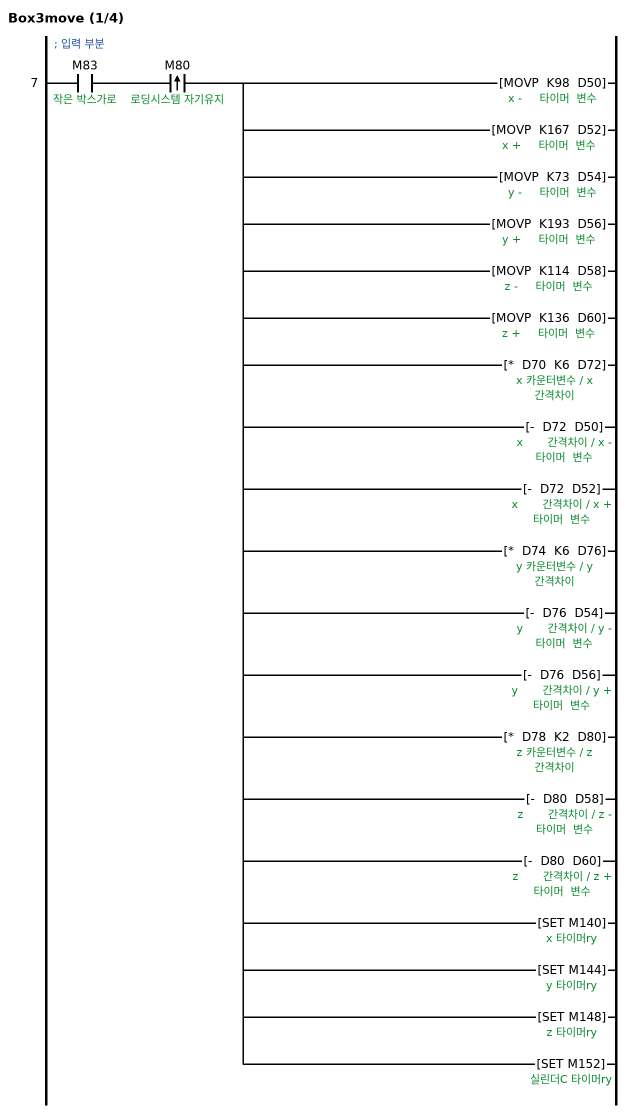
; 입력 부분
7     LD      M83  ; 작은 박스가로
      ANDP    M80  ; 로딩시스템 자기유지
      MOVP    K98 D50  ; x -     타이머  변수
      MOVP    K167 D52  ; x +     타이머  변수
      MOVP    K73 D54  ; y -     타이머  변수
      MOVP    K193 D56  ; y +     타이머  변수
      MOVP    K114 D58  ; z -     타이머  변수
      MOVP    K136 D60  ; z +     타이머  변수
      *       D70 K6 D72  ; x 카운터변수 / x       간격차이
      -       D72 D50
      -       D72 D52
      *       D74 K6 D76  ; y 카운터변수 / y       간격차이
      -       D76 D54
      -       D76 D56
      *       D78 K2 D80  ; z 카운터변수 / z       간격차이
      -       D80 D58
      -       D80 D60
      SET     M140  ; x 타이머ry
      SET     M144  ; y 타이머ry
      SET     M148  ; z 타이머ry
      SET     M152  ; 실린더C 타이머ry
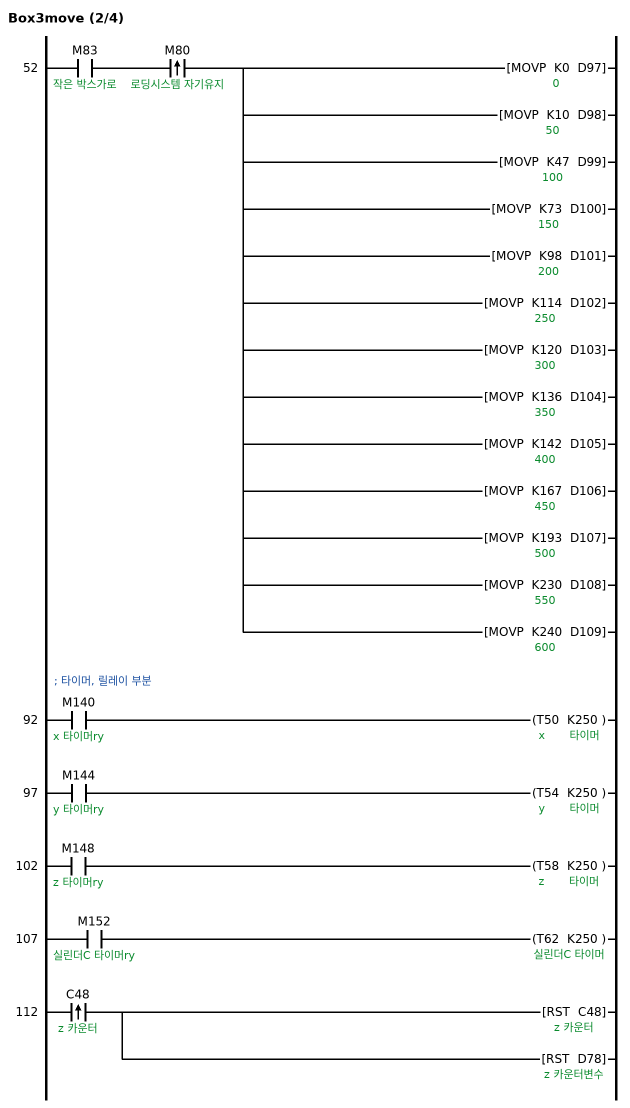
52    LD      M83  ; 작은 박스가로
      ANDP    M80  ; 로딩시스템 자기유지
      MOVP    K0 D97  ; 0
      MOVP    K10 D98  ; 50
      MOVP    K47 D99  ; 100
      MOVP    K73 D100  ; 150
      MOVP    K98 D101  ; 200
      MOVP    K114 D102  ; 250
      MOVP    K120 D103  ; 300
      MOVP    K136 D104  ; 350
      MOVP    K142 D105  ; 400
      MOVP    K167 D106  ; 450
      MOVP    K193 D107  ; 500
      MOVP    K230 D108  ; 550
      MOVP    K240 D109  ; 600
; 타이머, 릴레이 부분
92    LD      M140  ; x 타이머ry
      OUT     T50 K250  ; x       타이머
97    LD      M144  ; y 타이머ry
      OUT     T54 K250  ; y       타이머
102   LD      M148  ; z 타이머ry
      OUT     T58 K250  ; z       타이머
107   LD      M152  ; 실린더C 타이머ry
      OUT     T62 K250  ; 실린더C 타이머
112   LDP     C48  ; z 카운터
      RST     C48  ; z 카운터
      RST     D78  ; z 카운터변수
